TYPE stackerUnLoadImage :
STRUCT
	xLock1_lock 	        	   : imageIO := ( stIO  := Stations.sUnloadHmiIO.x_Lock1_lock,
									   image  		:= ADR(Global.INPUT_IMAGE),
									   iType  		:= ioType.INPUT_BIT,
									   iByte 		:= 17,
									   iBit  		:= 0 );	
									   
   xLock1_unlock				: imageIO := ( stIO   := Stations.sUnloadHmiIO.x_Lock1_unlock,
									   image 		  := ADR(Global.INPUT_IMAGE),
									   iType  		  := ioType.INPUT_BIT,
									   iByte 		  := 17,
									   iBit   		  := 1 );

    xLock2_lock 				: imageIO := ( stIO   := Stations.sUnloadHmiIO.x_Lock2_lock,
									   image  		  := ADR(Global.INPUT_IMAGE),
									   iType  		  := ioType.INPUT_BIT,
									   iByte 		  := 17,
									   iBit   		  := 2 );
									  
    xLock2_unlock 				: imageIO := ( stIO   := Stations.sUnloadHmiIO.x_Lock2_unlock,
									   image  		  := ADR(Global.INPUT_IMAGE),
									   iType  		  := ioType.INPUT_BIT,
									   iByte 		  := 17,
									   iBit   		  := 3 );

    xPalletOnTop 				: imageIO := ( stIO   := Stations.sUnloadHmiIO.x_PalletOnTop,
									   image  		  := ADR(Global.INPUT_IMAGE),
									   iType  		  := ioType.INPUT_BIT,
									   iByte 		  := 17,
									   iBit   		  := 6 );

    xPalletFix_lock 				: imageIO := ( stIO   := Stations.sUnloadHmiIO.x_PalletFix_lock,
									   image  		  := ADR(Global.INPUT_IMAGE),
									   iType  		  := ioType.INPUT_BIT,
									   iByte 		  := 17,
									   iBit   		  := 4 );

    xPalletFix_unlock 				: imageIO := ( stIO   := Stations.sUnloadHmiIO.x_PalletFix_unlock,
									   image  		  := ADR(Global.INPUT_IMAGE),
									   iType  		  := ioType.INPUT_BIT,
									   iByte 		  := 17,
									   iBit   		  := 5 );

    yLocks_lock 				: imageIO := ( stIO   := Stations.sUnloadHmiIO.y_Locks_lock,
									   image  		  := ADR(Global.OUTPUT_IMAGE),
									   iType  		  := ioType.OUTPUT_BIT,
									   iByte 		  := 151,
									   iBit   		  := 3 ); 

    yLocks_unlock 				: imageIO := ( stIO   := Stations.sUnloadHmiIO.y_Locks_unlock,
									   image  		  := ADR(Global.OUTPUT_IMAGE),
									   iType  		  := ioType.OUTPUT_BIT,
									   iByte 		  := 151,
									   iBit   		  := 2 ); 
 
    yPalletFix_lock 				: imageIO := ( stIO   := Stations.sUnloadHmiIO.y_PalletFix_lock,
									   image  		  := ADR(Global.OUTPUT_IMAGE),
									   iType  		  := ioType.OUTPUT_BIT,
									   iByte 		  := 151,
									   iBit   		  := 6 ); 
									   
    yPalletFix_unlock 				: imageIO := ( stIO   := Stations.sUnloadHmiIO.y_PalletFix_unlock,
									   image  		  := ADR(Global.OUTPUT_IMAGE),
									   iType  		  := ioType.OUTPUT_BIT,
									   iByte 		  := 151,
									   iBit   		  := 7 ); 
								
END_STRUCT
END_TYPE

(* stored: Version 1.1.0.1, ProductVersion 3.1.4024.3
   DUT stackerUnLoadImage: Id {7fc89de5-e988-4b65-83d9-c447efbc9098} *)
